ABB RobotStudio station: rdl.rsstn

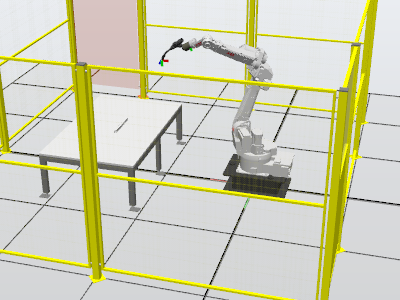
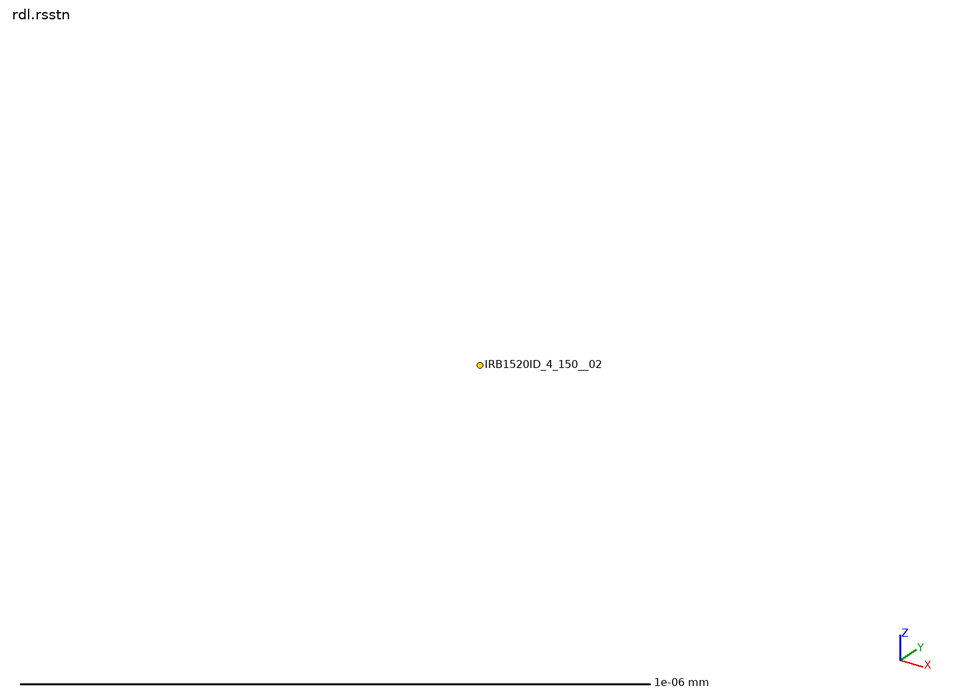
[picture v1: parts stored in the station drawn from their meshes, with robot base, taught points and paths (robot models come from the ABB library and are not in the file)]
Station Station (saved by RobotStudio 25.5.11605.0)
Controller rdl, task T_ROB1: task frame (RAPID world) sits at (0, 0, 205) mm in the station
Controller rdl
  mechanical unit ROB_1: IRB1520ID_4_150__02, 6 joints, base frame (0, 0, 0) mm
Layout (positions relative to the parent item):
  - RA_MTG4000_22 [mechanism, from %ABB.RobotStudio.Models.ArcWelding%\Fronius_Robacta_MTG4000_22deg.rslib] at (643.33, 235.52, 1605.87) mm, rotated rx -130.29 ry 39.35 rz -118.26 deg
  - IRB1520ID_4_150__02 [mechanism, from %ABB.RobotStudio.Models.IRB1520ID%\IRB1520ID_4_150_G_02.rslib] at (0, 0, 205) mm; joint values [0.4644, -0.3455, -0.1013, -0.4587, 1.0675, -0.27] (rad or m)
  - Robotpedestal1400_H240 [part, from Equipment\Robot Pedestal 1400 H240.rslib] at (-30, 0, 0) mm
  - Fence [graphiccomponentgroup]
    - Segment 1 [part], size 169.7 x 169.7 x 2000 mm
    - Segment 2 [part], size 169.7 x 2056 x 2000 mm
  - Fence_2 [graphiccomponentgroup]
    - Segment 1 [part], size 169.7 x 169.7 x 2000 mm
    - Segment 2 [part], size 1565.8 x 169.7 x 2000 mm
    - Segment 2 [part], size 1565.8 x 169.7 x 2000 mm
  - Fence_3 [graphiccomponentgroup]
    - Segment 1 [part], size 169.7 x 169.7 x 2000 mm
    - Segment 2 [part], size 169.7 x 2076.7 x 2000 mm
    - Segment 2 [part], size 169.7 x 2076.7 x 2000 mm
  - Fence_4 [graphiccomponentgroup]
    - Segment 1 [part], size 169.7 x 169.7 x 2000 mm
    - Segment 2 [part], size 2068.1 x 169.7 x 2000 mm
    - Segment 2 [part], size 2068.1 x 169.7 x 2000 mm
  - Fence_5 [graphiccomponentgroup]
    - Segment 1 [part], size 169.7 x 169.7 x 2000 mm
    - Segment 2 [part], size 169.7 x 1104.5 x 2000 mm
  - Fence_6 [graphiccomponentgroup]
    - Segment 1 [part], size 169.7 x 169.7 x 2000 mm
    - Segment 2 [part], size 169.7 x 1104.5 x 2000 mm
  - Fence_7 [graphiccomponentgroup]
    - Segment 1 [part], size 169.7 x 169.7 x 2000 mm
    - Segment 2 [part], size 169.7 x 1104.5 x 2000 mm
  - Fence_8 [graphiccomponentgroup]
    - Segment 1 [part], size 169.7 x 169.7 x 2000 mm
    - Segment 2 [part], size 1079.7 x 169.7 x 2000 mm
  - Table [part], size 1100 x 1635 x 500 mm
  - A-00677209-00_--E [graphiccomponentgroup] at (1701.18, 200, 677.03) mm, rotated rx 0 ry 0.1 rz 0 deg
    - A-00677226-00.12 [graphiccomponentgroup]
      - P039334634.1 [part], size 32 x 18 x 18 mm
    - A-00677216-00.7 [graphiccomponentgroup]
      - P039334633.2 [part], size 20 x 342 x 30 mm
    - A-00677226-00.11 [graphiccomponentgroup] at (0, 59, 0) mm
      - P039334634.1 [part], size 32 x 18 x 18 mm
Attachment: RA_MTG4000_22 is attached to IRB1520ID_4_150__02 / Link6
Targets, tools, work objects and paths stored in the station, written as RAPID:
! task T_ROB1
MODULE CalibData
  PERS tooldata torch:=[TRUE,[[20.31,0,363.689],[0.948464781,0,0.316882565,0]],[1,[0,0,1],[1,0,0,0],0,0,0]];
ENDMODULE

